(* IEC 61131-3 sources: mect_apps/TPAC1008_02_AB/RTU_test_PLC, 6 files *)

(* ---- Crosstable.gvl ---- *)
VAR_GLOBAL
errors_can AT %QD0.772:DINT;
errors_all AT %QD0.776:DINT;
min_latency_ms AT %QD0.780:DINT;
max_latency_ms AT %QD0.784:DINT;
Addr_node01 AT %IW0.800:UINT;
Life_node01 AT %IW0.804:UINT;
AnInCnf_1_node01 AT %QW0.808:UINT;
AnInCnf_2_node01 AT %QW0.812:UINT;
ValAi1_node01 AT %IW0.816:INT;
ValAi2_node01 AT %IW0.820:INT;
DigDir_1_node01 AT %QX0.824.0:BOOL;
DigDir_2_node01 AT %QX0.828.0:BOOL;
DigDir_3_node01 AT %QX0.832.0:BOOL;
DigDir_4_node01 AT %QX0.836.0:BOOL;
DigDir_5_node01 AT %QX0.840.0:BOOL;
DigDir_6_node01 AT %QX0.844.0:BOOL;
DigDir_7_node01 AT %QX0.848.0:BOOL;
DigDir_8_node01 AT %QX0.852.0:BOOL;
DigIn_2_node01 AT %IX0.856.0:BOOL;
DigIn_3_node01 AT %IX0.860.0:BOOL;
DigIn_6_node01 AT %IX0.864.0:BOOL;
DigIn_7_node01 AT %IX0.868.0:BOOL;
DigOut_1_node01 AT %QX0.872.0:BOOL;
DigOut_4_node01 AT %QX0.876.0:BOOL;
DigOut_5_node01 AT %QX0.880.0:BOOL;
DigOut_8_node01 AT %QX0.884.0:BOOL;
latency_01_ms AT %QD0.892:DINT;
min_latency_01_m AT %QD0.896:DINT;
max_latency_01_m AT %QD0.900:DINT;
errors_01 AT %QD0.908:DINT;
Addr_node02 AT %IW0.920:UINT;
Life_node02 AT %IW0.924:UINT;
AnInCnf_1_node02 AT %QW0.928:UINT;
AnInCnf_2_node02 AT %QW0.932:UINT;
ValAi1_node02 AT %IW0.936:INT;
ValAi2_node02 AT %IW0.940:INT;
DigDir_1_node02 AT %QX0.944.0:BOOL;
DigDir_2_node02 AT %QX0.948.0:BOOL;
DigDir_3_node02 AT %QX0.952.0:BOOL;
DigDir_4_node02 AT %QX0.956.0:BOOL;
DigDir_5_node02 AT %QX0.960.0:BOOL;
DigDir_6_node02 AT %QX0.964.0:BOOL;
DigDir_7_node02 AT %QX0.968.0:BOOL;
DigDir_8_node02 AT %QX0.972.0:BOOL;
DigIn_2_node02 AT %IX0.976.0:BOOL;
DigIn_3_node02 AT %IX0.980.0:BOOL;
DigIn_6_node02 AT %IX0.984.0:BOOL;
DigIn_7_node02 AT %IX0.988.0:BOOL;
DigOut_1_node02 AT %QX0.992.0:BOOL;
DigOut_4_node02 AT %QX0.996.0:BOOL;
DigOut_5_node02 AT %QX0.1000.0:BOOL;
DigOut_8_node02 AT %QX0.1004.0:BOOL;
latency_02_ms AT %QD0.1012:DINT;
min_latency_02_m AT %QD0.1016:DINT;
max_latency_02_m AT %QD0.1020:DINT;
errors_02 AT %QD0.1028:DINT;
Addr_node03 AT %IW0.1040:UINT;
Life_node03 AT %IW0.1044:UINT;
AnInCnf_1_node03 AT %QW0.1048:UINT;
AnInCnf_2_node03 AT %QW0.1052:UINT;
ValAi1_node03 AT %IW0.1056:INT;
ValAi2_node03 AT %IW0.1060:INT;
DigDir_1_node03 AT %QX0.1064.0:BOOL;
DigDir_2_node03 AT %QX0.1068.0:BOOL;
DigDir_3_node03 AT %QX0.1072.0:BOOL;
DigDir_4_node03 AT %QX0.1076.0:BOOL;
DigDir_5_node03 AT %QX0.1080.0:BOOL;
DigDir_6_node03 AT %QX0.1084.0:BOOL;
DigDir_7_node03 AT %QX0.1088.0:BOOL;
DigDir_8_node03 AT %QX0.1092.0:BOOL;
DigIn_2_node03 AT %IX0.1096.0:BOOL;
DigIn_3_node03 AT %IX0.1100.0:BOOL;
DigIn_6_node03 AT %IX0.1104.0:BOOL;
DigIn_7_node03 AT %IX0.1108.0:BOOL;
DigOut_1_node03 AT %QX0.1112.0:BOOL;
DigOut_4_node03 AT %QX0.1116.0:BOOL;
DigOut_5_node03 AT %QX0.1120.0:BOOL;
DigOut_8_node03 AT %QX0.1124.0:BOOL;
latency_03_ms AT %QD0.1132:DINT;
min_latency_03_m AT %QD0.1136:DINT;
max_latency_03_m AT %QD0.1140:DINT;
errors_03 AT %QD0.1148:DINT;
Addr_node04 AT %IW0.1160:UINT;
Life_node04 AT %IW0.1164:UINT;
AnInCnf_1_node04 AT %QW0.1168:UINT;
AnInCnf_2_node04 AT %QW0.1172:UINT;
ValAi1_node04 AT %IW0.1176:INT;
ValAi2_node04 AT %IW0.1180:INT;
DigDir_1_node04 AT %QX0.1184.0:BOOL;
DigDir_2_node04 AT %QX0.1188.0:BOOL;
DigDir_3_node04 AT %QX0.1192.0:BOOL;
DigDir_4_node04 AT %QX0.1196.0:BOOL;
DigDir_5_node04 AT %QX0.1200.0:BOOL;
DigDir_6_node04 AT %QX0.1204.0:BOOL;
DigDir_7_node04 AT %QX0.1208.0:BOOL;
DigDir_8_node04 AT %QX0.1212.0:BOOL;
DigIn_2_node04 AT %IX0.1216.0:BOOL;
DigIn_3_node04 AT %IX0.1220.0:BOOL;
DigIn_6_node04 AT %IX0.1224.0:BOOL;
DigIn_7_node04 AT %IX0.1228.0:BOOL;
DigOut_1_node04 AT %QX0.1232.0:BOOL;
DigOut_4_node04 AT %QX0.1236.0:BOOL;
DigOut_5_node04 AT %QX0.1240.0:BOOL;
DigOut_8_node04 AT %QX0.1244.0:BOOL;
latency_04_ms AT %QD0.1252:DINT;
min_latency_04_m AT %QD0.1256:DINT;
max_latency_04_m AT %QD0.1260:DINT;
errors_04 AT %QD0.1268:DINT;
Addr_node05 AT %IW0.1280:UINT;
Life_node05 AT %IW0.1284:UINT;
AnInCnf_1_node05 AT %QW0.1288:UINT;
AnInCnf_2_node05 AT %QW0.1292:UINT;
ValAi1_node05 AT %IW0.1296:INT;
ValAi2_node05 AT %IW0.1300:INT;
DigDir_1_node05 AT %QX0.1304.0:BOOL;
DigDir_2_node05 AT %QX0.1308.0:BOOL;
DigDir_3_node05 AT %QX0.1312.0:BOOL;
DigDir_4_node05 AT %QX0.1316.0:BOOL;
DigDir_5_node05 AT %QX0.1320.0:BOOL;
DigDir_6_node05 AT %QX0.1324.0:BOOL;
DigDir_7_node05 AT %QX0.1328.0:BOOL;
DigDir_8_node05 AT %QX0.1332.0:BOOL;
DigIn_2_node05 AT %IX0.1336.0:BOOL;
DigIn_3_node05 AT %IX0.1340.0:BOOL;
DigIn_6_node05 AT %IX0.1344.0:BOOL;
DigIn_7_node05 AT %IX0.1348.0:BOOL;
DigOut_1_node05 AT %QX0.1352.0:BOOL;
DigOut_4_node05 AT %QX0.1356.0:BOOL;
DigOut_5_node05 AT %QX0.1360.0:BOOL;
DigOut_8_node05 AT %QX0.1364.0:BOOL;
latency_05_ms AT %QD0.1372:DINT;
min_latency_05_m AT %QD0.1376:DINT;
max_latency_05_m AT %QD0.1380:DINT;
errors_05 AT %QD0.1388:DINT;
Addr_node06 AT %IW0.1400:UINT;
Life_node06 AT %IW0.1404:UINT;
AnInCnf_1_node06 AT %QW0.1408:UINT;
AnInCnf_2_node06 AT %QW0.1412:UINT;
ValAi1_node06 AT %IW0.1416:INT;
ValAi2_node06 AT %IW0.1420:INT;
DigDir_1_node06 AT %QX0.1424.0:BOOL;
DigDir_2_node06 AT %QX0.1428.0:BOOL;
DigDir_3_node06 AT %QX0.1432.0:BOOL;
DigDir_4_node06 AT %QX0.1436.0:BOOL;
DigDir_5_node06 AT %QX0.1440.0:BOOL;
DigDir_6_node06 AT %QX0.1444.0:BOOL;
DigDir_7_node06 AT %QX0.1448.0:BOOL;
DigDir_8_node06 AT %QX0.1452.0:BOOL;
DigIn_2_node06 AT %IX0.1456.0:BOOL;
DigIn_3_node06 AT %IX0.1460.0:BOOL;
DigIn_6_node06 AT %IX0.1464.0:BOOL;
DigIn_7_node06 AT %IX0.1468.0:BOOL;
DigOut_1_node06 AT %QX0.1472.0:BOOL;
DigOut_4_node06 AT %QX0.1476.0:BOOL;
DigOut_5_node06 AT %QX0.1480.0:BOOL;
DigOut_8_node06 AT %QX0.1484.0:BOOL;
latency_06_ms AT %QD0.1492:DINT;
min_latency_06_m AT %QD0.1496:DINT;
max_latency_06_m AT %QD0.1500:DINT;
errors_06 AT %QD0.1508:DINT;
Addr_node07 AT %IW0.1520:UINT;
Life_node07 AT %IW0.1524:UINT;
AnInCnf_1_node07 AT %QW0.1528:UINT;
AnInCnf_2_node07 AT %QW0.1532:UINT;
ValAi1_node07 AT %IW0.1536:INT;
ValAi2_node07 AT %IW0.1540:INT;
DigDir_1_node07 AT %QX0.1544.0:BOOL;
DigDir_2_node07 AT %QX0.1548.0:BOOL;
DigDir_3_node07 AT %QX0.1552.0:BOOL;
DigDir_4_node07 AT %QX0.1556.0:BOOL;
DigDir_5_node07 AT %QX0.1560.0:BOOL;
DigDir_6_node07 AT %QX0.1564.0:BOOL;
DigDir_7_node07 AT %QX0.1568.0:BOOL;
DigDir_8_node07 AT %QX0.1572.0:BOOL;
DigIn_2_node07 AT %IX0.1576.0:BOOL;
DigIn_3_node07 AT %IX0.1580.0:BOOL;
DigIn_6_node07 AT %IX0.1584.0:BOOL;
DigIn_7_node07 AT %IX0.1588.0:BOOL;
DigOut_1_node07 AT %QX0.1592.0:BOOL;
DigOut_4_node07 AT %QX0.1596.0:BOOL;
DigOut_5_node07 AT %QX0.1600.0:BOOL;
DigOut_8_node07 AT %QX0.1604.0:BOOL;
latency_07_ms AT %QD0.1612:DINT;
min_latency_07_m AT %QD0.1616:DINT;
max_latency_07_m AT %QD0.1620:DINT;
errors_07 AT %QD0.1628:DINT;
Addr_node08 AT %IW0.1640:UINT;
Life_node08 AT %IW0.1644:UINT;
AnInCnf_1_node08 AT %QW0.1648:UINT;
AnInCnf_2_node08 AT %QW0.1652:UINT;
ValAi1_node08 AT %IW0.1656:INT;
ValAi2_node08 AT %IW0.1660:INT;
DigDir_1_node08 AT %QX0.1664.0:BOOL;
DigDir_2_node08 AT %QX0.1668.0:BOOL;
DigDir_3_node08 AT %QX0.1672.0:BOOL;
DigDir_4_node08 AT %QX0.1676.0:BOOL;
DigDir_5_node08 AT %QX0.1680.0:BOOL;
DigDir_6_node08 AT %QX0.1684.0:BOOL;
DigDir_7_node08 AT %QX0.1688.0:BOOL;
DigDir_8_node08 AT %QX0.1692.0:BOOL;
DigIn_2_node08 AT %IX0.1696.0:BOOL;
DigIn_3_node08 AT %IX0.1700.0:BOOL;
DigIn_6_node08 AT %IX0.1704.0:BOOL;
DigIn_7_node08 AT %IX0.1708.0:BOOL;
DigOut_1_node08 AT %QX0.1712.0:BOOL;
DigOut_4_node08 AT %QX0.1716.0:BOOL;
DigOut_5_node08 AT %QX0.1720.0:BOOL;
DigOut_8_node08 AT %QX0.1724.0:BOOL;
latency_08_ms AT %QD0.1732:DINT;
min_latency_08_m AT %QD0.1736:DINT;
max_latency_08_m AT %QD0.1740:DINT;
errors_08 AT %QD0.1748:DINT;
Addr_node09 AT %IW0.1760:UINT;
Life_node09 AT %IW0.1764:UINT;
AnInCnf_1_node09 AT %QW0.1768:UINT;
AnInCnf_2_node09 AT %QW0.1772:UINT;
ValAi1_node09 AT %IW0.1776:INT;
ValAi2_node09 AT %IW0.1780:INT;
DigDir_1_node09 AT %QX0.1784.0:BOOL;
DigDir_2_node09 AT %QX0.1788.0:BOOL;
DigDir_3_node09 AT %QX0.1792.0:BOOL;
DigDir_4_node09 AT %QX0.1796.0:BOOL;
DigDir_5_node09 AT %QX0.1800.0:BOOL;
DigDir_6_node09 AT %QX0.1804.0:BOOL;
DigDir_7_node09 AT %QX0.1808.0:BOOL;
DigDir_8_node09 AT %QX0.1812.0:BOOL;
DigIn_2_node09 AT %IX0.1816.0:BOOL;
DigIn_3_node09 AT %IX0.1820.0:BOOL;
DigIn_6_node09 AT %IX0.1824.0:BOOL;
DigIn_7_node09 AT %IX0.1828.0:BOOL;
DigOut_1_node09 AT %QX0.1832.0:BOOL;
DigOut_4_node09 AT %QX0.1836.0:BOOL;
DigOut_5_node09 AT %QX0.1840.0:BOOL;
DigOut_8_node09 AT %QX0.1844.0:BOOL;
latency_09_ms AT %QD0.1852:DINT;
min_latency_09_m AT %QD0.1856:DINT;
max_latency_09_m AT %QD0.1860:DINT;
errors_09 AT %QD0.1868:DINT;
Addr_node10 AT %IW0.1880:UINT;
Life_node10 AT %IW0.1884:UINT;
AnInCnf_1_node10 AT %QW0.1888:UINT;
AnInCnf_2_node10 AT %QW0.1892:UINT;
ValAi1_node10 AT %IW0.1896:INT;
ValAi2_node10 AT %IW0.1900:INT;
DigDir_1_node10 AT %QX0.1904.0:BOOL;
DigDir_2_node10 AT %QX0.1908.0:BOOL;
DigDir_3_node10 AT %QX0.1912.0:BOOL;
DigDir_4_node10 AT %QX0.1916.0:BOOL;
DigDir_5_node10 AT %QX0.1920.0:BOOL;
DigDir_6_node10 AT %QX0.1924.0:BOOL;
DigDir_7_node10 AT %QX0.1928.0:BOOL;
DigDir_8_node10 AT %QX0.1932.0:BOOL;
DigIn_2_node10 AT %IX0.1936.0:BOOL;
DigIn_3_node10 AT %IX0.1940.0:BOOL;
DigIn_6_node10 AT %IX0.1944.0:BOOL;
DigIn_7_node10 AT %IX0.1948.0:BOOL;
DigOut_1_node10 AT %QX0.1952.0:BOOL;
DigOut_4_node10 AT %QX0.1956.0:BOOL;
DigOut_5_node10 AT %QX0.1960.0:BOOL;
DigOut_8_node10 AT %QX0.1964.0:BOOL;
latency_10_ms AT %QD0.1972:DINT;
min_latency_10_m AT %QD0.1976:DINT;
max_latency_10_m AT %QD0.1980:DINT;
errors_10 AT %QD0.1988:DINT;
Addr_node11 AT %IW0.2000:UINT;
Life_node11 AT %IW0.2004:UINT;
AnInCnf_1_node11 AT %QW0.2008:UINT;
AnInCnf_2_node11 AT %QW0.2012:UINT;
ValAi1_node11 AT %IW0.2016:INT;
ValAi2_node11 AT %IW0.2020:INT;
DigDir_1_node11 AT %QX0.2024.0:BOOL;
DigDir_2_node11 AT %QX0.2028.0:BOOL;
DigDir_3_node11 AT %QX0.2032.0:BOOL;
DigDir_4_node11 AT %QX0.2036.0:BOOL;
DigDir_5_node11 AT %QX0.2040.0:BOOL;
DigDir_6_node11 AT %QX0.2044.0:BOOL;
DigDir_7_node11 AT %QX0.2048.0:BOOL;
DigDir_8_node11 AT %QX0.2052.0:BOOL;
DigIn_2_node11 AT %IX0.2056.0:BOOL;
DigIn_3_node11 AT %IX0.2060.0:BOOL;
DigIn_6_node11 AT %IX0.2064.0:BOOL;
DigIn_7_node11 AT %IX0.2068.0:BOOL;
DigOut_1_node11 AT %QX0.2072.0:BOOL;
DigOut_4_node11 AT %QX0.2076.0:BOOL;
DigOut_5_node11 AT %QX0.2080.0:BOOL;
DigOut_8_node11 AT %QX0.2084.0:BOOL;
latency_11_ms AT %QD0.2092:DINT;
min_latency_11_m AT %QD0.2096:DINT;
max_latency_11_m AT %QD0.2100:DINT;
errors_11 AT %QD0.2108:DINT;
Addr_node12 AT %IW0.2120:UINT;
Life_node12 AT %IW0.2124:UINT;
AnInCnf_1_node12 AT %QW0.2128:UINT;
AnInCnf_2_node12 AT %QW0.2132:UINT;
ValAi1_node12 AT %IW0.2136:INT;
ValAi2_node12 AT %IW0.2140:INT;
DigDir_1_node12 AT %QX0.2144.0:BOOL;
DigDir_2_node12 AT %QX0.2148.0:BOOL;
DigDir_3_node12 AT %QX0.2152.0:BOOL;
DigDir_4_node12 AT %QX0.2156.0:BOOL;
DigDir_5_node12 AT %QX0.2160.0:BOOL;
DigDir_6_node12 AT %QX0.2164.0:BOOL;
DigDir_7_node12 AT %QX0.2168.0:BOOL;
DigDir_8_node12 AT %QX0.2172.0:BOOL;
DigIn_2_node12 AT %IX0.2176.0:BOOL;
DigIn_3_node12 AT %IX0.2180.0:BOOL;
DigIn_6_node12 AT %IX0.2184.0:BOOL;
DigIn_7_node12 AT %IX0.2188.0:BOOL;
DigOut_1_node12 AT %QX0.2192.0:BOOL;
DigOut_4_node12 AT %QX0.2196.0:BOOL;
DigOut_5_node12 AT %QX0.2200.0:BOOL;
DigOut_8_node12 AT %QX0.2204.0:BOOL;
latency_12_ms AT %QD0.2212:DINT;
min_latency_12_m AT %QD0.2216:DINT;
max_latency_12_m AT %QD0.2220:DINT;
errors_12 AT %QD0.2228:DINT;
Addr_node13 AT %IW0.2240:UINT;
Life_node13 AT %IW0.2244:UINT;
AnInCnf_1_node13 AT %QW0.2248:UINT;
AnInCnf_2_node13 AT %QW0.2252:UINT;
ValAi1_node13 AT %IW0.2256:INT;
ValAi2_node13 AT %IW0.2260:INT;
DigDir_1_node13 AT %QX0.2264.0:BOOL;
DigDir_2_node13 AT %QX0.2268.0:BOOL;
DigDir_3_node13 AT %QX0.2272.0:BOOL;
DigDir_4_node13 AT %QX0.2276.0:BOOL;
DigDir_5_node13 AT %QX0.2280.0:BOOL;
DigDir_6_node13 AT %QX0.2284.0:BOOL;
DigDir_7_node13 AT %QX0.2288.0:BOOL;
DigDir_8_node13 AT %QX0.2292.0:BOOL;
DigIn_2_node13 AT %IX0.2296.0:BOOL;
DigIn_3_node13 AT %IX0.2300.0:BOOL;
DigIn_6_node13 AT %IX0.2304.0:BOOL;
DigIn_7_node13 AT %IX0.2308.0:BOOL;
DigOut_1_node13 AT %QX0.2312.0:BOOL;
DigOut_4_node13 AT %QX0.2316.0:BOOL;
DigOut_5_node13 AT %QX0.2320.0:BOOL;
DigOut_8_node13 AT %QX0.2324.0:BOOL;
latency_13_ms AT %QD0.2332:DINT;
min_latency_13_m AT %QD0.2336:DINT;
max_latency_13_m AT %QD0.2340:DINT;
errors_13 AT %QD0.2348:DINT;
Addr_node14 AT %IW0.2360:UINT;
Life_node14 AT %IW0.2364:UINT;
AnInCnf_1_node14 AT %QW0.2368:UINT;
AnInCnf_2_node14 AT %QW0.2372:UINT;
ValAi1_node14 AT %IW0.2376:INT;
ValAi2_node14 AT %IW0.2380:INT;
DigDir_1_node14 AT %QX0.2384.0:BOOL;
DigDir_2_node14 AT %QX0.2388.0:BOOL;
DigDir_3_node14 AT %QX0.2392.0:BOOL;
DigDir_4_node14 AT %QX0.2396.0:BOOL;
DigDir_5_node14 AT %QX0.2400.0:BOOL;
DigDir_6_node14 AT %QX0.2404.0:BOOL;
DigDir_7_node14 AT %QX0.2408.0:BOOL;
DigDir_8_node14 AT %QX0.2412.0:BOOL;
DigIn_2_node14 AT %IX0.2416.0:BOOL;
DigIn_3_node14 AT %IX0.2420.0:BOOL;
DigIn_6_node14 AT %IX0.2424.0:BOOL;
DigIn_7_node14 AT %IX0.2428.0:BOOL;
DigOut_1_node14 AT %QX0.2432.0:BOOL;
DigOut_4_node14 AT %QX0.2436.0:BOOL;
DigOut_5_node14 AT %QX0.2440.0:BOOL;
DigOut_8_node14 AT %QX0.2444.0:BOOL;
latency_14_ms AT %QD0.2452:DINT;
min_latency_14_m AT %QD0.2456:DINT;
max_latency_14_m AT %QD0.2460:DINT;
errors_14 AT %QD0.2468:DINT;
Addr_node15 AT %IW0.2480:UINT;
Life_node15 AT %IW0.2484:UINT;
AnInCnf_1_node15 AT %QW0.2488:UINT;
AnInCnf_2_node15 AT %QW0.2492:UINT;
ValAi1_node15 AT %IW0.2496:INT;
ValAi2_node15 AT %IW0.2500:INT;
DigDir_1_node15 AT %QX0.2504.0:BOOL;
DigDir_2_node15 AT %QX0.2508.0:BOOL;
DigDir_3_node15 AT %QX0.2512.0:BOOL;
DigDir_4_node15 AT %QX0.2516.0:BOOL;
DigDir_5_node15 AT %QX0.2520.0:BOOL;
DigDir_6_node15 AT %QX0.2524.0:BOOL;
DigDir_7_node15 AT %QX0.2528.0:BOOL;
DigDir_8_node15 AT %QX0.2532.0:BOOL;
DigIn_2_node15 AT %IX0.2536.0:BOOL;
DigIn_3_node15 AT %IX0.2540.0:BOOL;
DigIn_6_node15 AT %IX0.2544.0:BOOL;
DigIn_7_node15 AT %IX0.2548.0:BOOL;
DigOut_1_node15 AT %QX0.2552.0:BOOL;
DigOut_4_node15 AT %QX0.2556.0:BOOL;
DigOut_5_node15 AT %QX0.2560.0:BOOL;
DigOut_8_node15 AT %QX0.2564.0:BOOL;
latency_15_ms AT %QD0.2572:DINT;
min_latency_15_m AT %QD0.2576:DINT;
max_latency_15_m AT %QD0.2580:DINT;
errors_15 AT %QD0.2588:DINT;
Addr_node16 AT %IW0.2600:UINT;
Life_node16 AT %IW0.2604:UINT;
AnInCnf_1_node16 AT %QW0.2608:UINT;
AnInCnf_2_node16 AT %QW0.2612:UINT;
ValAi1_node16 AT %IW0.2616:INT;
ValAi2_node16 AT %IW0.2620:INT;
DigDir_1_node16 AT %QX0.2624.0:BOOL;
DigDir_2_node16 AT %QX0.2628.0:BOOL;
DigDir_3_node16 AT %QX0.2632.0:BOOL;
DigDir_4_node16 AT %QX0.2636.0:BOOL;
DigDir_5_node16 AT %QX0.2640.0:BOOL;
DigDir_6_node16 AT %QX0.2644.0:BOOL;
DigDir_7_node16 AT %QX0.2648.0:BOOL;
DigDir_8_node16 AT %QX0.2652.0:BOOL;
DigIn_2_node16 AT %IX0.2656.0:BOOL;
DigIn_3_node16 AT %IX0.2660.0:BOOL;
DigIn_6_node16 AT %IX0.2664.0:BOOL;
DigIn_7_node16 AT %IX0.2668.0:BOOL;
DigOut_1_node16 AT %QX0.2672.0:BOOL;
DigOut_4_node16 AT %QX0.2676.0:BOOL;
DigOut_5_node16 AT %QX0.2680.0:BOOL;
DigOut_8_node16 AT %QX0.2684.0:BOOL;
latency_16_ms AT %QD0.2692:DINT;
min_latency_16_m AT %QD0.2696:DINT;
max_latency_16_m AT %QD0.2700:DINT;
errors_16 AT %QD0.2708:DINT;
Addr_node17 AT %IW0.2720:UINT;
Life_node17 AT %IW0.2724:UINT;
AnInCnf_1_node17 AT %QW0.2728:UINT;
AnInCnf_2_node17 AT %QW0.2732:UINT;
ValAi1_node17 AT %IW0.2736:INT;
ValAi2_node17 AT %IW0.2740:INT;
DigDir_1_node17 AT %QX0.2744.0:BOOL;
DigDir_2_node17 AT %QX0.2748.0:BOOL;
DigDir_3_node17 AT %QX0.2752.0:BOOL;
DigDir_4_node17 AT %QX0.2756.0:BOOL;
DigDir_5_node17 AT %QX0.2760.0:BOOL;
DigDir_6_node17 AT %QX0.2764.0:BOOL;
DigDir_7_node17 AT %QX0.2768.0:BOOL;
DigDir_8_node17 AT %QX0.2772.0:BOOL;
DigIn_2_node17 AT %IX0.2776.0:BOOL;
DigIn_3_node17 AT %IX0.2780.0:BOOL;
DigIn_6_node17 AT %IX0.2784.0:BOOL;
DigIn_7_node17 AT %IX0.2788.0:BOOL;
DigOut_1_node17 AT %QX0.2792.0:BOOL;
DigOut_4_node17 AT %QX0.2796.0:BOOL;
DigOut_5_node17 AT %QX0.2800.0:BOOL;
DigOut_8_node17 AT %QX0.2804.0:BOOL;
latency_17_ms AT %QD0.2812:DINT;
min_latency_17_m AT %QD0.2816:DINT;
max_latency_17_m AT %QD0.2820:DINT;
errors_17 AT %QD0.2828:DINT;
Addr_node18 AT %IW0.2840:UINT;
Life_node18 AT %IW0.2844:UINT;
AnInCnf_1_node18 AT %QW0.2848:UINT;
AnInCnf_2_node18 AT %QW0.2852:UINT;
ValAi1_node18 AT %IW0.2856:INT;
ValAi2_node18 AT %IW0.2860:INT;
DigDir_1_node18 AT %QX0.2864.0:BOOL;
DigDir_2_node18 AT %QX0.2868.0:BOOL;
DigDir_3_node18 AT %QX0.2872.0:BOOL;
DigDir_4_node18 AT %QX0.2876.0:BOOL;
DigDir_5_node18 AT %QX0.2880.0:BOOL;
DigDir_6_node18 AT %QX0.2884.0:BOOL;
DigDir_7_node18 AT %QX0.2888.0:BOOL;
DigDir_8_node18 AT %QX0.2892.0:BOOL;
DigIn_2_node18 AT %IX0.2896.0:BOOL;
DigIn_3_node18 AT %IX0.2900.0:BOOL;
DigIn_6_node18 AT %IX0.2904.0:BOOL;
DigIn_7_node18 AT %IX0.2908.0:BOOL;
DigOut_1_node18 AT %QX0.2912.0:BOOL;
DigOut_4_node18 AT %QX0.2916.0:BOOL;
DigOut_5_node18 AT %QX0.2920.0:BOOL;
DigOut_8_node18 AT %QX0.2924.0:BOOL;
latency_18_ms AT %QD0.2932:DINT;
min_latency_18_m AT %QD0.2936:DINT;
max_latency_18_m AT %QD0.2940:DINT;
errors_18 AT %QD0.2948:DINT;
Addr_node19 AT %IW0.2960:UINT;
Life_node19 AT %IW0.2964:UINT;
AnInCnf_1_node19 AT %QW0.2968:UINT;
AnInCnf_2_node19 AT %QW0.2972:UINT;
ValAi1_node19 AT %IW0.2976:INT;
ValAi2_node19 AT %IW0.2980:INT;
DigDir_1_node19 AT %QX0.2984.0:BOOL;
DigDir_2_node19 AT %QX0.2988.0:BOOL;
DigDir_3_node19 AT %QX0.2992.0:BOOL;
DigDir_4_node19 AT %QX0.2996.0:BOOL;
DigDir_5_node19 AT %QX0.3000.0:BOOL;
DigDir_6_node19 AT %QX0.3004.0:BOOL;
DigDir_7_node19 AT %QX0.3008.0:BOOL;
DigDir_8_node19 AT %QX0.3012.0:BOOL;
DigIn_2_node19 AT %IX0.3016.0:BOOL;
DigIn_3_node19 AT %IX0.3020.0:BOOL;
DigIn_6_node19 AT %IX0.3024.0:BOOL;
DigIn_7_node19 AT %IX0.3028.0:BOOL;
DigOut_1_node19 AT %QX0.3032.0:BOOL;
DigOut_4_node19 AT %QX0.3036.0:BOOL;
DigOut_5_node19 AT %QX0.3040.0:BOOL;
DigOut_8_node19 AT %QX0.3044.0:BOOL;
latency_19_ms AT %QD0.3052:DINT;
min_latency_19_m AT %QD0.3056:DINT;
max_latency_19_m AT %QD0.3060:DINT;
errors_19 AT %QD0.3068:DINT;
Addr_node20 AT %IW0.3080:UINT;
Life_node20 AT %IW0.3084:UINT;
AnInCnf_1_node20 AT %QW0.3088:UINT;
AnInCnf_2_node20 AT %QW0.3092:UINT;
ValAi1_node20 AT %IW0.3096:INT;
ValAi2_node20 AT %IW0.3100:INT;
DigDir_1_node20 AT %QX0.3104.0:BOOL;
DigDir_2_node20 AT %QX0.3108.0:BOOL;
DigDir_3_node20 AT %QX0.3112.0:BOOL;
DigDir_4_node20 AT %QX0.3116.0:BOOL;
DigDir_5_node20 AT %QX0.3120.0:BOOL;
DigDir_6_node20 AT %QX0.3124.0:BOOL;
DigDir_7_node20 AT %QX0.3128.0:BOOL;
DigDir_8_node20 AT %QX0.3132.0:BOOL;
DigIn_2_node20 AT %IX0.3136.0:BOOL;
DigIn_3_node20 AT %IX0.3140.0:BOOL;
DigIn_6_node20 AT %IX0.3144.0:BOOL;
DigIn_7_node20 AT %IX0.3148.0:BOOL;
DigOut_1_node20 AT %QX0.3152.0:BOOL;
DigOut_4_node20 AT %QX0.3156.0:BOOL;
DigOut_5_node20 AT %QX0.3160.0:BOOL;
DigOut_8_node20 AT %QX0.3164.0:BOOL;
latency_20_ms AT %QD0.3172:DINT;
min_latency_20_m AT %QD0.3176:DINT;
max_latency_20_m AT %QD0.3180:DINT;
errors_20 AT %QD0.3188:DINT;
Addr_node21 AT %IW0.3200:UINT;
Life_node21 AT %IW0.3204:UINT;
AnInCnf_1_node21 AT %QW0.3208:UINT;
AnInCnf_2_node21 AT %QW0.3212:UINT;
ValAi1_node21 AT %IW0.3216:INT;
ValAi2_node21 AT %IW0.3220:INT;
DigDir_1_node21 AT %QX0.3224.0:BOOL;
DigDir_2_node21 AT %QX0.3228.0:BOOL;
DigDir_3_node21 AT %QX0.3232.0:BOOL;
DigDir_4_node21 AT %QX0.3236.0:BOOL;
DigDir_5_node21 AT %QX0.3240.0:BOOL;
DigDir_6_node21 AT %QX0.3244.0:BOOL;
DigDir_7_node21 AT %QX0.3248.0:BOOL;
DigDir_8_node21 AT %QX0.3252.0:BOOL;
DigIn_2_node21 AT %IX0.3256.0:BOOL;
DigIn_3_node21 AT %IX0.3260.0:BOOL;
DigIn_6_node21 AT %IX0.3264.0:BOOL;
DigIn_7_node21 AT %IX0.3268.0:BOOL;
DigOut_1_node21 AT %QX0.3272.0:BOOL;
DigOut_4_node21 AT %QX0.3276.0:BOOL;
DigOut_5_node21 AT %QX0.3280.0:BOOL;
DigOut_8_node21 AT %QX0.3284.0:BOOL;
latency_21_ms AT %QD0.3292:DINT;
min_latency_21_m AT %QD0.3296:DINT;
max_latency_21_m AT %QD0.3300:DINT;
errors_21 AT %QD0.3308:DINT;
Addr_node22 AT %IW0.3320:UINT;
Life_node22 AT %IW0.3324:UINT;
AnInCnf_1_node22 AT %QW0.3328:UINT;
AnInCnf_2_node22 AT %QW0.3332:UINT;
ValAi1_node22 AT %IW0.3336:INT;
ValAi2_node22 AT %IW0.3340:INT;
DigDir_1_node22 AT %QX0.3344.0:BOOL;
DigDir_2_node22 AT %QX0.3348.0:BOOL;
DigDir_3_node22 AT %QX0.3352.0:BOOL;
DigDir_4_node22 AT %QX0.3356.0:BOOL;
DigDir_5_node22 AT %QX0.3360.0:BOOL;
DigDir_6_node22 AT %QX0.3364.0:BOOL;
DigDir_7_node22 AT %QX0.3368.0:BOOL;
DigDir_8_node22 AT %QX0.3372.0:BOOL;
DigIn_2_node22 AT %IX0.3376.0:BOOL;
DigIn_3_node22 AT %IX0.3380.0:BOOL;
DigIn_6_node22 AT %IX0.3384.0:BOOL;
DigIn_7_node22 AT %IX0.3388.0:BOOL;
DigOut_1_node22 AT %QX0.3392.0:BOOL;
DigOut_4_node22 AT %QX0.3396.0:BOOL;
DigOut_5_node22 AT %QX0.3400.0:BOOL;
DigOut_8_node22 AT %QX0.3404.0:BOOL;
latency_22_ms AT %QD0.3412:DINT;
min_latency_22_m AT %QD0.3416:DINT;
max_latency_22_m AT %QD0.3420:DINT;
errors_22 AT %QD0.3428:DINT;
Addr_node23 AT %IW0.3440:UINT;
Life_node23 AT %IW0.3444:UINT;
AnInCnf_1_node23 AT %QW0.3448:UINT;
AnInCnf_2_node23 AT %QW0.3452:UINT;
ValAi1_node23 AT %IW0.3456:INT;
ValAi2_node23 AT %IW0.3460:INT;
DigDir_1_node23 AT %QX0.3464.0:BOOL;
DigDir_2_node23 AT %QX0.3468.0:BOOL;
DigDir_3_node23 AT %QX0.3472.0:BOOL;
DigDir_4_node23 AT %QX0.3476.0:BOOL;
DigDir_5_node23 AT %QX0.3480.0:BOOL;
DigDir_6_node23 AT %QX0.3484.0:BOOL;
DigDir_7_node23 AT %QX0.3488.0:BOOL;
DigDir_8_node23 AT %QX0.3492.0:BOOL;
DigIn_2_node23 AT %IX0.3496.0:BOOL;
DigIn_3_node23 AT %IX0.3500.0:BOOL;
DigIn_6_node23 AT %IX0.3504.0:BOOL;
DigIn_7_node23 AT %IX0.3508.0:BOOL;
DigOut_1_node23 AT %QX0.3512.0:BOOL;
DigOut_4_node23 AT %QX0.3516.0:BOOL;
DigOut_5_node23 AT %QX0.3520.0:BOOL;
DigOut_8_node23 AT %QX0.3524.0:BOOL;
latency_23_ms AT %QD0.3532:DINT;
min_latency_23_m AT %QD0.3536:DINT;
max_latency_23_m AT %QD0.3540:DINT;
errors_23 AT %QD0.3548:DINT;
Addr_node24 AT %IW0.3560:UINT;
Life_node24 AT %IW0.3564:UINT;
AnInCnf_1_node24 AT %QW0.3568:UINT;
AnInCnf_2_node24 AT %QW0.3572:UINT;
ValAi1_node24 AT %IW0.3576:INT;
ValAi2_node24 AT %IW0.3580:INT;
DigDir_1_node24 AT %QX0.3584.0:BOOL;
DigDir_2_node24 AT %QX0.3588.0:BOOL;
DigDir_3_node24 AT %QX0.3592.0:BOOL;
DigDir_4_node24 AT %QX0.3596.0:BOOL;
DigDir_5_node24 AT %QX0.3600.0:BOOL;
DigDir_6_node24 AT %QX0.3604.0:BOOL;
DigDir_7_node24 AT %QX0.3608.0:BOOL;
DigDir_8_node24 AT %QX0.3612.0:BOOL;
DigIn_2_node24 AT %IX0.3616.0:BOOL;
DigIn_3_node24 AT %IX0.3620.0:BOOL;
DigIn_6_node24 AT %IX0.3624.0:BOOL;
DigIn_7_node24 AT %IX0.3628.0:BOOL;
DigOut_1_node24 AT %QX0.3632.0:BOOL;
DigOut_4_node24 AT %QX0.3636.0:BOOL;
DigOut_5_node24 AT %QX0.3640.0:BOOL;
DigOut_8_node24 AT %QX0.3644.0:BOOL;
latency_24_ms AT %QD0.3652:DINT;
min_latency_24_m AT %QD0.3656:DINT;
max_latency_24_m AT %QD0.3660:DINT;
errors_24 AT %QD0.3668:DINT;
RTU0_TYPE_PORT AT %ID0.20000:UDINT;
RTU0_BAUDRATE AT %ID0.20004:UDINT;
RTU0_STATUS AT %ID0.20008:UDINT;
RTU0_READS AT %ID0.20012:UDINT;
RTU0_WRITES AT %ID0.20016:UDINT;
RTU0_TIMEOUTS AT %ID0.20020:UDINT;
RTU0_COMM_ERRORS AT %ID0.20024:UDINT;
RTU0_LAST_ERROR AT %ID0.20028:UDINT;
RTU0_WRITE_QUEUE AT %ID0.20032:UDINT;
RTU0_READ_QUEUE AT %ID0.20036:UDINT;
RTU1_TYPE_PORT AT %ID0.20040:UDINT;
RTU1_BAUDRATE AT %ID0.20044:UDINT;
RTU1_STATUS AT %ID0.20048:UDINT;
RTU1_READS AT %ID0.20052:UDINT;
RTU1_WRITES AT %ID0.20056:UDINT;
RTU1_TIMEOUTS AT %ID0.20060:UDINT;
RTU1_COMM_ERRORS AT %ID0.20064:UDINT;
RTU1_LAST_ERROR AT %ID0.20068:UDINT;
RTU1_WRITE_QUEUE AT %ID0.20072:UDINT;
RTU1_READ_QUEUE AT %ID0.20076:UDINT;
RTU3_TYPE_PORT AT %ID0.20080:UDINT;
RTU3_BAUDRATE AT %ID0.20084:UDINT;
RTU3_STATUS AT %ID0.20088:UDINT;
RTU3_READS AT %ID0.20092:UDINT;
RTU3_WRITES AT %ID0.20096:UDINT;
RTU3_TIMEOUTS AT %ID0.20100:UDINT;
RTU3_COMM_ERRORS AT %ID0.20104:UDINT;
RTU3_LAST_ERROR AT %ID0.20108:UDINT;
RTU3_WRITE_QUEUE AT %ID0.20112:UDINT;
RTU3_READ_QUEUE AT %ID0.20116:UDINT;
CAN0_TYPE_PORT AT %ID0.20120:UDINT;
CAN0_BAUDRATE AT %ID0.20124:UDINT;
CAN0_STATUS AT %ID0.20128:UDINT;
CAN0_READS AT %ID0.20132:UDINT;
CAN0_WRITES AT %ID0.20136:UDINT;
CAN0_TIMEOUTS AT %ID0.20140:UDINT;
CAN0_COMM_ERRORS AT %ID0.20144:UDINT;
CAN0_LAST_ERROR AT %ID0.20148:UDINT;
CAN0_WRITE_QUEUE AT %ID0.20152:UDINT;
CAN0_READ_QUEUE AT %ID0.20156:UDINT;
CAN1_TYPE_PORT AT %ID0.20160:UDINT;
CAN1_BAUDRATE AT %ID0.20164:UDINT;
CAN1_STATUS AT %ID0.20168:UDINT;
CAN1_READS AT %ID0.20172:UDINT;
CAN1_WRITES AT %ID0.20176:UDINT;
CAN1_TIMEOUTS AT %ID0.20180:UDINT;
CAN1_COMM_ERRORS AT %ID0.20184:UDINT;
CAN1_LAST_ERROR AT %ID0.20188:UDINT;
CAN1_WRITE_QUEUE AT %ID0.20192:UDINT;
CAN1_READ_QUEUE AT %ID0.20196:UDINT;
TCPS_TYPE_PORT AT %ID0.20200:UDINT;
TCPS_IP_ADDRESS AT %ID0.20204:UDINT;
TCPS_STATUS AT %ID0.20208:UDINT;
TCPS_READS AT %ID0.20212:UDINT;
TCPS_WRITES AT %ID0.20216:UDINT;
TCPS_TIMEOUTS AT %ID0.20220:UDINT;
TCPS_COMM_ERRORS AT %ID0.20224:UDINT;
TCPS_LAST_ERROR AT %ID0.20228:UDINT;
TCPS_WRITE_QUEUE AT %ID0.20232:UDINT;
TCPS_READ_QUEUE AT %ID0.20236:UDINT;
TCP0_TYPE_PORT AT %ID0.20240:UDINT;
TCP0_IP_ADDRESS AT %ID0.20244:UDINT;
TCP0_STATUS AT %ID0.20248:UDINT;
TCP0_READS AT %ID0.20252:UDINT;
TCP0_WRITES AT %ID0.20256:UDINT;
TCP0_TIMEOUTS AT %ID0.20260:UDINT;
TCP0_COMM_ERRORS AT %ID0.20264:UDINT;
TCP0_LAST_ERROR AT %ID0.20268:UDINT;
TCP0_WRITE_QUEUE AT %ID0.20272:UDINT;
TCP0_READ_QUEUE AT %ID0.20276:UDINT;
TCP1_TYPE_PORT AT %ID0.20280:UDINT;
TCP1_IP_ADDRESS AT %ID0.20284:UDINT;
TCP1_STATUS AT %ID0.20288:UDINT;
TCP1_READS AT %ID0.20292:UDINT;
TCP1_WRITES AT %ID0.20296:UDINT;
TCP1_TIMEOUTS AT %ID0.20300:UDINT;
TCP1_COMM_ERRORS AT %ID0.20304:UDINT;
TCP1_LAST_ERROR AT %ID0.20308:UDINT;
TCP1_WRITE_QUEUE AT %ID0.20312:UDINT;
TCP1_READ_QUEUE AT %ID0.20316:UDINT;
TCP2_TYPE_PORT AT %ID0.20320:UDINT;
TCP2_IP_ADDRESS AT %ID0.20324:UDINT;
TCP2_STATUS AT %ID0.20328:UDINT;
TCP2_READS AT %ID0.20332:UDINT;
TCP2_WRITES AT %ID0.20336:UDINT;
TCP2_TIMEOUTS AT %ID0.20340:UDINT;
TCP2_COMM_ERRORS AT %ID0.20344:UDINT;
TCP2_LAST_ERROR AT %ID0.20348:UDINT;
TCP2_WRITE_QUEUE AT %ID0.20352:UDINT;
TCP2_READ_QUEUE AT %ID0.20356:UDINT;
TCP3_TYPE_PORT AT %ID0.20360:UDINT;
TCP3_IP_ADDRESS AT %ID0.20364:UDINT;
TCP3_STATUS AT %ID0.20368:UDINT;
TCP3_READS AT %ID0.20372:UDINT;
TCP3_WRITES AT %ID0.20376:UDINT;
TCP3_TIMEOUTS AT %ID0.20380:UDINT;
TCP3_COMM_ERRORS AT %ID0.20384:UDINT;
TCP3_LAST_ERROR AT %ID0.20388:UDINT;
TCP3_WRITE_QUEUE AT %ID0.20392:UDINT;
TCP3_READ_QUEUE AT %ID0.20396:UDINT;
TCP4_TYPE_PORT AT %ID0.20400:UDINT;
TCP4_IP_ADDRESS AT %ID0.20404:UDINT;
TCP4_STATUS AT %ID0.20408:UDINT;
TCP4_READS AT %ID0.20412:UDINT;
TCP4_WRITES AT %ID0.20416:UDINT;
TCP4_TIMEOUTS AT %ID0.20420:UDINT;
TCP4_COMM_ERRORS AT %ID0.20424:UDINT;
TCP4_LAST_ERROR AT %ID0.20428:UDINT;
TCP4_WRITE_QUEUE AT %ID0.20432:UDINT;
TCP4_READ_QUEUE AT %ID0.20436:UDINT;
TCP5_TYPE_PORT AT %ID0.20440:UDINT;
TCP5_IP_ADDRESS AT %ID0.20444:UDINT;
TCP5_STATUS AT %ID0.20448:UDINT;
TCP5_READS AT %ID0.20452:UDINT;
TCP5_WRITES AT %ID0.20456:UDINT;
TCP5_TIMEOUTS AT %ID0.20460:UDINT;
TCP5_COMM_ERRORS AT %ID0.20464:UDINT;
TCP5_LAST_ERROR AT %ID0.20468:UDINT;
TCP5_WRITE_QUEUE AT %ID0.20472:UDINT;
TCP5_READ_QUEUE AT %ID0.20476:UDINT;
TCP6_TYPE_PORT AT %ID0.20480:UDINT;
TCP6_IP_ADDRESS AT %ID0.20484:UDINT;
TCP6_STATUS AT %ID0.20488:UDINT;
TCP6_READS AT %ID0.20492:UDINT;
TCP6_WRITES AT %ID0.20496:UDINT;
TCP6_TIMEOUTS AT %ID0.20500:UDINT;
TCP6_COMM_ERRORS AT %ID0.20504:UDINT;
TCP6_LAST_ERROR AT %ID0.20508:UDINT;
TCP6_WRITE_QUEUE AT %ID0.20512:UDINT;
TCP6_READ_QUEUE AT %ID0.20516:UDINT;
TCP7_TYPE_PORT AT %ID0.20520:UDINT;
TCP7_IP_ADDRESS AT %ID0.20524:UDINT;
TCP7_STATUS AT %ID0.20528:UDINT;
TCP7_READS AT %ID0.20532:UDINT;
TCP7_WRITES AT %ID0.20536:UDINT;
TCP7_TIMEOUTS AT %ID0.20540:UDINT;
TCP7_COMM_ERRORS AT %ID0.20544:UDINT;
TCP7_LAST_ERROR AT %ID0.20548:UDINT;
TCP7_WRITE_QUEUE AT %ID0.20552:UDINT;
TCP7_READ_QUEUE AT %ID0.20556:UDINT;
TCP8_TYPE_PORT AT %ID0.20560:UDINT;
TCP8_IP_ADDRESS AT %ID0.20564:UDINT;
TCP8_STATUS AT %ID0.20568:UDINT;
TCP8_READS AT %ID0.20572:UDINT;
TCP8_WRITES AT %ID0.20576:UDINT;
TCP8_TIMEOUTS AT %ID0.20580:UDINT;
TCP8_COMM_ERRORS AT %ID0.20584:UDINT;
TCP8_LAST_ERROR AT %ID0.20588:UDINT;
TCP8_WRITE_QUEUE AT %ID0.20592:UDINT;
TCP8_READ_QUEUE AT %ID0.20596:UDINT;
TCP9_TYPE_PORT AT %ID0.20600:UDINT;
TCP9_IP_ADDRESS AT %ID0.20604:UDINT;
TCP9_STATUS AT %ID0.20608:UDINT;
TCP9_READS AT %ID0.20612:UDINT;
TCP9_WRITES AT %ID0.20616:UDINT;
TCP9_TIMEOUTS AT %ID0.20620:UDINT;
TCP9_COMM_ERRORS AT %ID0.20624:UDINT;
TCP9_LAST_ERROR AT %ID0.20628:UDINT;
TCP9_WRITE_QUEUE AT %ID0.20632:UDINT;
TCP9_READ_QUEUE AT %ID0.20636:UDINT;
NODE_01_DEV_NODE AT %ID0.20688:UDINT;
NODE_01_STATUS AT %ID0.20692:UDINT;
NODE_02_DEV_NODE AT %ID0.20696:UDINT;
NODE_02_STATUS AT %ID0.20700:UDINT;
NODE_03_DEV_NODE AT %ID0.20704:UDINT;
NODE_03_STATUS AT %ID0.20708:UDINT;
NODE_04_DEV_NODE AT %ID0.20712:UDINT;
NODE_04_STATUS AT %ID0.20716:UDINT;
NODE_05_DEV_NODE AT %ID0.20720:UDINT;
NODE_05_STATUS AT %ID0.20724:UDINT;
NODE_06_DEV_NODE AT %ID0.20728:UDINT;
NODE_06_STATUS AT %ID0.20732:UDINT;
NODE_07_DEV_NODE AT %ID0.20736:UDINT;
NODE_07_STATUS AT %ID0.20740:UDINT;
NODE_08_DEV_NODE AT %ID0.20744:UDINT;
NODE_08_STATUS AT %ID0.20748:UDINT;
NODE_09_DEV_NODE AT %ID0.20752:UDINT;
NODE_09_STATUS AT %ID0.20756:UDINT;
NODE_10_DEV_NODE AT %ID0.20760:UDINT;
NODE_10_STATUS AT %ID0.20764:UDINT;
NODE_11_DEV_NODE AT %ID0.20768:UDINT;
NODE_11_STATUS AT %ID0.20772:UDINT;
NODE_12_DEV_NODE AT %ID0.20776:UDINT;
NODE_12_STATUS AT %ID0.20780:UDINT;
NODE_13_DEV_NODE AT %ID0.20784:UDINT;
NODE_13_STATUS AT %ID0.20788:UDINT;
NODE_14_DEV_NODE AT %ID0.20792:UDINT;
NODE_14_STATUS AT %ID0.20796:UDINT;
NODE_15_DEV_NODE AT %ID0.20800:UDINT;
NODE_15_STATUS AT %ID0.20804:UDINT;
NODE_16_DEV_NODE AT %ID0.20808:UDINT;
NODE_16_STATUS AT %ID0.20812:UDINT;
NODE_17_DEV_NODE AT %ID0.20816:UDINT;
NODE_17_STATUS AT %ID0.20820:UDINT;
NODE_18_DEV_NODE AT %ID0.20824:UDINT;
NODE_18_STATUS AT %ID0.20828:UDINT;
NODE_19_DEV_NODE AT %ID0.20832:UDINT;
NODE_19_STATUS AT %ID0.20836:UDINT;
NODE_20_DEV_NODE AT %ID0.20840:UDINT;
NODE_20_STATUS AT %ID0.20844:UDINT;
NODE_21_DEV_NODE AT %ID0.20848:UDINT;
NODE_21_STATUS AT %ID0.20852:UDINT;
NODE_22_DEV_NODE AT %ID0.20856:UDINT;
NODE_22_STATUS AT %ID0.20860:UDINT;
NODE_23_DEV_NODE AT %ID0.20864:UDINT;
NODE_23_STATUS AT %ID0.20868:UDINT;
NODE_24_DEV_NODE AT %ID0.20872:UDINT;
NODE_24_STATUS AT %ID0.20876:UDINT;
PLC_DigIn_1 AT %IX0.21200.0:BOOL;
PLC_DigIn_2 AT %IX0.21204.0:BOOL;
PLC_DigIn_3 AT %IX0.21208.0:BOOL;
PLC_DigIn_4 AT %IX0.21212.0:BOOL;
PLC_DigIn_5 AT %IX0.21216.0:BOOL;
PLC_DigIn_6 AT %IX0.21220.0:BOOL;
PLC_DigIn_7 AT %IX0.21224.0:BOOL;
PLC_DigIn_8 AT %IX0.21228.0:BOOL;
PLC_Reserved_1 AT %IX0.21232.0:BOOL;
PLC_DigOut_1 AT %QX0.21236.0:BOOL;
PLC_DigOut_2 AT %QX0.21240.0:BOOL;
PLC_DigOut_3 AT %QX0.21244.0:BOOL;
PLC_DigOut_4 AT %QX0.21248.0:BOOL;
PLC_DigOut_5 AT %QX0.21252.0:BOOL;
PLC_DigOut_6 AT %QX0.21256.0:BOOL;
PLC_DigOut_7 AT %QX0.21260.0:BOOL;
PLC_DigOut_8 AT %QX0.21264.0:BOOL;
PLC_DigOut_9 AT %QX0.21268.0:BOOL;
PLC_DigOut_10 AT %QX0.21272.0:BOOL;
PLC_DigOut_11 AT %QX0.21276.0:BOOL;
PLC_DigOut_12 AT %QX0.21280.0:BOOL;
PLC_Hwconf AT %IW0.21284:UINT;
PLC_Revisione AT %IW0.21288:UINT;
PLC_StatusReg AT %IW0.21292:UINT;
PLC_Heartbeat AT %IW0.21296:UINT;
PLC_AnIn_1 AT %IW0.21300:INT;
PLC_AnIn_2 AT %IW0.21304:INT;
PLC_AnIn_3 AT %IW0.21308:INT;
PLC_AnIn_4 AT %IW0.21312:INT;
PLC_EncoderCo_Lo AT %IW0.21316:UINT;
PLC_EncoderCo_Hi AT %IW0.21320:UINT;
PLC_CaptureT1_Lo AT %IW0.21324:UINT;
PLC_CaptureT1_Hi AT %IW0.21328:UINT;
PLC_CaptureT2_Lo AT %IW0.21332:UINT;
PLC_CaptureT2_Hi AT %IW0.21336:UINT;
PLC_RPM AT %IW0.21340:UINT;
PLC_Tamb AT %IW0.21344:INT;
PLC_EnableEnc AT %QW0.21348:UINT;
PLC_ResetCount AT %QW0.21352:UINT;
PLC_AnInConf_1 AT %QW0.21356:UINT;
PLC_AnInConf_2 AT %QW0.21360:UINT;
PLC_AnInConf_3 AT %QW0.21364:UINT;
PLC_AnInConf_4 AT %QW0.21368:UINT;
PLC_AnOutConf_1 AT %QW0.21372:UINT;
PLC_AnOutConf_2 AT %QW0.21376:UINT;
PLC_Reserved_2 AT %QW0.21380:UINT;
PLC_Reserved_3 AT %QW0.21384:UINT;
PLC_AnOut_1 AT %QW0.21388:INT;
PLC_AnOut_2 AT %QW0.21392:INT;
PLC_Reserved_4 AT %QW0.21396:INT;
PLC_Reserved_5 AT %QW0.21400:INT;
PLC_FiltAnIn_1 AT %QW0.21404:UINT;
PLC_FiltAnIn_2 AT %QW0.21408:UINT;
PLC_FiltAnIn_3 AT %QW0.21412:UINT;
PLC_FiltAnIn_4 AT %QW0.21416:UINT;
CH0_NETRUN AT %IX0.21428.0:BOOL;
CH0_NETGOOD AT %IX0.21432.0:BOOL;
CH0_NETERR AT %ID0.21436:UDINT;
CH0_NETRST AT %QX0.21440.0:BOOL;
CH0_NETDIS AT %QX0.21444.0:BOOL;
CH0_01_NODERUN AT %IX0.21448.0:BOOL;
CH0_01_NODEGOOD AT %IX0.21452.0:BOOL;
CH0_01_NODEERR AT %ID0.21456:UDINT;
CH0_01_NODERST AT %QX0.21460.0:BOOL;
CH0_01_NODEDIS AT %QX0.21464.0:BOOL;
PLC_time AT %ID0.21560:REAL;
PLC_timeMin AT %ID0.21564:REAL;
PLC_timeMax AT %ID0.21568:REAL;
PLC_timeWin AT %QD0.21572:REAL;
PLC_Version AT %IW0.21576:UINT;
PLC_EngineStatus AT %IW0.21580:UINT;
PLC_ResetValues AT %QX0.21584.0:BOOL;
PLC_buzzerOn AT %QX0.21588.0:BOOL;
END_VAR

(* ---- set_min_dint.st ---- *)
(*[[
]]*)
FUNCTION set_min_dint
VAR_IN_OUT
    A : DINT;
END_VAR
VAR_INPUT
    B : DINT;
END_VAR

	if A < 0 or B < A then
		A := B;
	end_if;

END_FUNCTION

(* ---- Fast.st ---- *)
(*[[
]]*)
PROGRAM Fast
#import "Crosstable.gvl"
#import "Resource1.gvl"
VAR

END_VAR

;

END_PROGRAM

(* ---- Init.st ---- *)
(*[[
]]*)
PROGRAM Init
#import "Crosstable.gvl"
#import "Resource1.gvl"

Conf1_node01 :=1;
Conf1_node02 :=1;
Conf1_node03 :=1;
Conf1_node04 :=1;
Conf1_node05 :=1;
Conf1_node06 :=1;
Conf1_node07 :=1;
Conf1_node08 :=1;
Conf1_node09 :=1;
Conf1_node10 :=1;
Conf1_node11 :=1;
Conf1_node12 :=1;
Conf1_node13 :=1;
Conf1_node14 :=1;
Conf1_node15 :=1;
Conf1_node16 :=1;
Conf1_node17 :=1;
Conf1_node18 :=1;
Conf1_node19 :=1;
Conf1_node20 :=1;
Conf1_node21 :=1;
Conf1_node22 :=1;
Conf1_node23 :=1;
Conf1_node24 :=1;

Conf2_node01 :=1;
Conf2_node02 :=1;
Conf2_node03 :=1;
Conf2_node04 :=1;
Conf2_node05 :=1;
Conf2_node06 :=1;
Conf2_node07 :=1;
Conf2_node08 :=1;
Conf2_node09 :=1;
Conf2_node10 :=1;
Conf2_node11 :=1;
Conf2_node12 :=1;
Conf2_node13 :=1;
Conf2_node14 :=1;
Conf2_node15 :=1;
Conf2_node16 :=1;
Conf2_node17 :=1;
Conf2_node18 :=1;
Conf2_node19 :=1;
Conf2_node20 :=1;
Conf2_node21 :=1;
Conf2_node22 :=1;
Conf2_node23 :=1;
Conf2_node24 :=1;

Conf3_node01 :=1;
Conf3_node02 :=1;
Conf3_node03 :=1;
Conf3_node04 :=1;
Conf3_node05 :=1;
Conf3_node06 :=1;
Conf3_node07 :=1;
Conf3_node08 :=1;
Conf3_node09 :=1;
Conf3_node10 :=1;
Conf3_node11 :=1;
Conf3_node12 :=1;
Conf3_node13 :=1;
Conf3_node14 :=1;
Conf3_node15 :=1;
Conf3_node16 :=1;
Conf3_node17 :=1;
Conf3_node18 :=1;
Conf3_node19 :=1;
Conf3_node20 :=1;
Conf3_node21 :=1;
Conf3_node22 :=1;
Conf3_node23 :=1;
Conf3_node24 :=1;

Conf4_node01 :=1;
Conf4_node02 :=1;
Conf4_node03 :=1;
Conf4_node04 :=1;
Conf4_node05 :=1;
Conf4_node06 :=1;
Conf4_node07 :=1;
Conf4_node08 :=1;
Conf4_node09 :=1;
Conf4_node10 :=1;
Conf4_node11 :=1;
Conf4_node12 :=1;
Conf4_node13 :=1;
Conf4_node14 :=1;
Conf4_node15 :=1;
Conf4_node16 :=1;
Conf4_node17 :=1;
Conf4_node18 :=1;
Conf4_node19 :=1;
Conf4_node20 :=1;
Conf4_node21 :=1;
Conf4_node22 :=1;
Conf4_node23 :=1;
Conf4_node24 :=1;

ConfAi1_node01 := 2;
ConfAi1_node02 := 2;
ConfAi1_node03 := 2;
ConfAi1_node04 := 2;
ConfAi1_node05 := 2;
ConfAi1_node06 := 2;
ConfAi1_node07 := 2;
ConfAi1_node08 := 2;
ConfAi1_node09 := 2;
ConfAi1_node10 := 2;
ConfAi1_node11 := 2;
ConfAi1_node12 := 2;
ConfAi1_node13 := 2;
ConfAi1_node14 := 2;
ConfAi1_node15 := 2;
ConfAi1_node16 := 2;
ConfAi1_node17 := 2;
ConfAi1_node18 := 2;
ConfAi1_node19 := 2;
ConfAi1_node20 := 2;
ConfAi1_node21 := 2;
ConfAi1_node22 := 2;
ConfAi1_node23 := 2;
ConfAi1_node24 := 2;

ConfAi2_node01 := 2;
ConfAi2_node02 := 2;
ConfAi2_node03 := 2;
ConfAi2_node04 := 2;
ConfAi2_node05 := 2;
ConfAi2_node06 := 2;
ConfAi2_node07 := 2;
ConfAi2_node08 := 2;
ConfAi2_node09 := 2;
ConfAi2_node10 := 2;
ConfAi2_node11 := 2;
ConfAi2_node12 := 2;
ConfAi2_node13 := 2;
ConfAi2_node14 := 2;
ConfAi2_node15 := 2;
ConfAi2_node16 := 2;
ConfAi2_node17 := 2;
ConfAi2_node18 := 2;
ConfAi2_node19 := 2;
ConfAi2_node20 := 2;
ConfAi2_node21 := 2;
ConfAi2_node22 := 2;
ConfAi2_node23 := 2;
ConfAi2_node24 := 2;

END_PROGRAM

(* ---- Normal.st ---- *)
(*[[
]]*)
PROGRAM Normal
#import "Crosstable.gvl"
#import "Resource1.gvl"
VAR
	counter : uint := 0;
	onoff : bool := true;
	first : bool := true;
	timer : TON;
	value : bool := true;
	timer_ms : UINT := 0;
	do_second_loop : bool := false;

END_VAR

	(* increment timer *)
	timer_ms := timer_ms + 50;

	(* check can status *)
	if CH0_01_NODERUN = false then
		if not first then
			errors_can := errors_can + 1;
		end_if;
 	    return;
	end_if;

	(* init *)
	if first then
		first := false;

		(* 0. init analog outputs *)
		PLC_AnOutConf_1 := 2;
		PLC_AnOutConf_2 := 2;
		PLC_AnOut_1 := 0;
		PLC_AnOut_2 := 0;

		errors_can := 0;

		(* 1. reset latency errors *)
		errors_01 := 0;
		errors_02 := 0;
		errors_03 := 0;
		errors_04 := 0;
		errors_05 := 0;
		errors_06 := 0;
		errors_07 := 0;
		errors_08 := 0;
		errors_09 := 0;
		errors_10 := 0;
		errors_11 := 0;
		errors_12 := 0;
		errors_13 := 0;
		errors_14 := 0;
		errors_15 := 0;
		errors_16 := 0;
		errors_17 := 0;
		errors_18 := 0;
		errors_19 := 0;
		errors_20 := 0;
		errors_21 := 0;
		errors_22 := 0;
		errors_23 := 0;
		errors_24 := 0;

		(* 2. reset latency timer *)
		timer_ms := 0;

		(* 3. reset latencies, ... *)
		latency_01_ms := 0;
		latency_02_ms := 0;
		latency_03_ms := 0;
		latency_04_ms := 0;
		latency_05_ms := 0;
		latency_06_ms := 0;
		latency_07_ms := 0;
		latency_08_ms := 0;
		latency_09_ms := 0;
		latency_10_ms := 0;
		latency_11_ms := 0;
		latency_12_ms := 0;
		latency_13_ms := 0;
		latency_14_ms := 0;
		latency_15_ms := 0;
		latency_16_ms := 0;
		latency_17_ms := 0;
		latency_18_ms := 0;
		latency_19_ms := 0;
		latency_20_ms := 0;
		latency_21_ms := 0;
		latency_22_ms := 0;
		latency_23_ms := 0;
		latency_24_ms := 0;

		min_latency_01_m := 0;
		min_latency_02_m := 0;
		min_latency_03_m := 0;
		min_latency_04_m := 0;
		min_latency_05_m := 0;
		min_latency_06_m := 0;
		min_latency_07_m := 0;
		min_latency_08_m := 0;
		min_latency_09_m := 0;
		min_latency_10_m := 0;
		min_latency_11_m := 0;
		min_latency_12_m := 0;
		min_latency_13_m := 0;
		min_latency_14_m := 0;
		min_latency_15_m := 0;
		min_latency_16_m := 0;
		min_latency_17_m := 0;
		min_latency_18_m := 0;
		min_latency_19_m := 0;
		min_latency_20_m := 0;
		min_latency_21_m := 0;
		min_latency_22_m := 0;
		min_latency_23_m := 0;
		min_latency_24_m := 0;

		max_latency_01_m := 0;
		max_latency_02_m := 0;
		max_latency_03_m := 0;
		max_latency_04_m := 0;
		max_latency_05_m := 0;
		max_latency_06_m := 0;
		max_latency_07_m := 0;
		max_latency_08_m := 0;
		max_latency_09_m := 0;
		max_latency_10_m := 0;
		max_latency_11_m := 0;
		max_latency_12_m := 0;
		max_latency_13_m := 0;
		max_latency_14_m := 0;
		max_latency_15_m := 0;
		max_latency_16_m := 0;
		max_latency_17_m := 0;
		max_latency_18_m := 0;
		max_latency_19_m := 0;
		max_latency_20_m := 0;
		max_latency_21_m := 0;
		max_latency_22_m := 0;
		max_latency_23_m := 0;
		max_latency_24_m := 0;

		(* 4. set first output values *)
		value := true;
		PLC_DigOut_1 := true;
		PLC_AnOut_1 := 900;
		PLC_AnOut_2 := 100;

	end_if;

	timer (IN := true, PT := T#4s);

	(* FIRST/LAST STEP *)
	if timer.q = true then

		(* 0. rearm timer *)
		timer (IN := false);

		(* 1. check latency errors *)
		if latency_01_ms = 0 then
			errors_01 := errors_01 + 1;
		end_if;
		if latency_02_ms = 0 then
			errors_02 := errors_02 + 1;
		end_if;
		if latency_03_ms = 0 then
			errors_03 := errors_03 + 1;
		end_if;
		if latency_04_ms = 0 then
			errors_04 := errors_04 + 1;
		end_if;
		if latency_05_ms = 0 then
			errors_05 := errors_05 + 1;
		end_if;
		if latency_06_ms = 0 then
			errors_06 := errors_06 + 1;
		end_if;
		if latency_07_ms = 0 then
			errors_07 := errors_07 + 1;
		end_if;
		if latency_08_ms = 0 then
			errors_08 := errors_08 + 1;
		end_if;
		if latency_09_ms = 0 then
			errors_09 := errors_09 + 1;
		end_if;
		if latency_10_ms = 0 then
			errors_10 := errors_10 + 1;
		end_if;
		if latency_11_ms = 0 then
			errors_11 := errors_11 + 1;
		end_if;
		if latency_12_ms = 0 then
			errors_12 := errors_12 + 1;
		end_if;
		if latency_13_ms = 0 then
			errors_13 := errors_13 + 1;
		end_if;
		if latency_14_ms = 0 then
			errors_14 := errors_14 + 1;
		end_if;
		if latency_15_ms = 0 then
			errors_15 := errors_15 + 1;
		end_if;
		if latency_16_ms = 0 then
			errors_16 := errors_16 + 1;
		end_if;
		if latency_17_ms = 0 then
			errors_17 := errors_17 + 1;
		end_if;
		if latency_18_ms = 0 then
			errors_18 := errors_18 + 1;
		end_if;
		if latency_19_ms = 0 then
			errors_19 := errors_19 + 1;
		end_if;
		if latency_20_ms = 0 then
			errors_20 := errors_20 + 1;
		end_if;
		if latency_21_ms = 0 then
			errors_21 := errors_21 + 1;
		end_if;
		if latency_22_ms = 0 then
			errors_22 := errors_22 + 1;
		end_if;
		if latency_23_ms = 0 then
			errors_23 := errors_23 + 1;
		end_if;
		if latency_24_ms = 0 then
			errors_24 := errors_24 + 1;
		end_if;

		(* 2. reset latency timer *)
		timer_ms := 0;

		(* 3. reset latencies, ... *)
	    latency_01_ms := 0;
		latency_02_ms := 0;
		latency_03_ms := 0;
		latency_04_ms := 0;
		latency_05_ms := 0;
		latency_06_ms := 0;
		latency_07_ms := 0;
		latency_08_ms := 0;
		latency_09_ms := 0;
		latency_10_ms := 0;
		latency_11_ms := 0;
		latency_12_ms := 0;
		latency_13_ms := 0;
		latency_14_ms := 0;
		latency_15_ms := 0;
		latency_16_ms := 0;
		latency_17_ms := 0;
		latency_18_ms := 0;
		latency_19_ms := 0;
		latency_20_ms := 0;
		latency_21_ms := 0;
		latency_22_ms := 0;
		latency_23_ms := 0;
		latency_24_ms := 0;

		(* 4. set new output value *)
		value := not value;
		PLC_DigOut_1 := value;
		if value then
			PLC_AnOut_1 := 900;
			PLC_AnOut_2 := 100;
		else
			PLC_AnOut_1 := 100;
			PLC_AnOut_2 := 900;
		end_if;

	(* OTHER STEPS *)
	else

		(* for each node: latency from TPAC:DigOut_1 to NODE:DigIn_7 to NODE:DigOut_8 *)

		if latency_01_ms = 0 and DigIn_7_node01 = value then
			(* measure the latency *)
		    latency_01_ms := timer_ms;
			if max_latency_01_m < timer_ms then
				max_latency_01_m := timer_ms;
			end_if;
			if min_latency_01_m > timer_ms or min_latency_01_m = 0 then
				min_latency_01_m := timer_ms;
			end_if;
			(* write the output *)
			DigOut_8_node01 := value;
		end_if;
		if latency_02_ms = 0 and DigIn_7_node02 = value then
			(* measure the latency *)
		    latency_02_ms := timer_ms;
			if max_latency_02_m < timer_ms then
				max_latency_02_m := timer_ms;
			end_if;
			if min_latency_02_m > timer_ms or min_latency_02_m = 0 then
				min_latency_02_m := timer_ms;
			end_if;
			(* write the output *)
			DigOut_8_node02 := value;
		end_if;
		if latency_03_ms = 0 and DigIn_7_node03 = value then
			(* measure the latency *)
		    latency_03_ms := timer_ms;
			if max_latency_03_m < timer_ms then
				max_latency_03_m := timer_ms;
			end_if;
			if min_latency_03_m > timer_ms or min_latency_03_m = 0 then
				min_latency_03_m := timer_ms;
			end_if;
			(* write the output *)
			DigOut_8_node03 := value;
		end_if;
		if latency_04_ms = 0 and DigIn_7_node04 = value then
			(* measure the latency *)
		    latency_04_ms := timer_ms;
			if max_latency_04_m < timer_ms then
				max_latency_04_m := timer_ms;
			end_if;
			if min_latency_04_m > timer_ms or min_latency_04_m = 0 then
				min_latency_04_m := timer_ms;
			end_if;
			(* write the output *)
			DigOut_8_node04 := value;
		end_if;
		if latency_05_ms = 0 and DigIn_7_node05 = value then
			(* measure the latency *)
		    latency_05_ms := timer_ms;
			if max_latency_05_m < timer_ms then
				max_latency_05_m := timer_ms;
			end_if;
			if min_latency_05_m > timer_ms or min_latency_05_m = 0 then
				min_latency_05_m := timer_ms;
			end_if;
			(* write the output *)
			DigOut_8_node05 := value;
		end_if;
		if latency_06_ms = 0 and DigIn_7_node06 = value then
			(* measure the latency *)
		    latency_06_ms := timer_ms;
			if max_latency_06_m < timer_ms then
				max_latency_06_m := timer_ms;
			end_if;
			if min_latency_06_m > timer_ms or min_latency_06_m = 0 then
				min_latency_06_m := timer_ms;
			end_if;
			(* write the output *)
			DigOut_8_node06 := value;
		end_if;
		if latency_07_ms = 0 and DigIn_7_node07 = value then
			(* measure the latency *)
		    latency_07_ms := timer_ms;
			if max_latency_07_m < timer_ms then
				max_latency_07_m := timer_ms;
			end_if;
			if min_latency_07_m > timer_ms or min_latency_07_m = 0 then
				min_latency_07_m := timer_ms;
			end_if;
			(* write the output *)
			DigOut_8_node07 := value;
		end_if;
		if latency_08_ms = 0 and DigIn_7_node08 = value then
			(* measure the latency *)
		    latency_08_ms := timer_ms;
			if max_latency_08_m < timer_ms then
				max_latency_08_m := timer_ms;
			end_if;
			if min_latency_08_m > timer_ms or min_latency_08_m = 0 then
				min_latency_08_m := timer_ms;
			end_if;
			(* write the output *)
			DigOut_8_node08 := value;
		end_if;
		if latency_09_ms = 0 and DigIn_7_node09 = value then
			(* measure the latency *)
		    latency_09_ms := timer_ms;
			if max_latency_09_m < timer_ms then
				max_latency_09_m := timer_ms;
			end_if;
			if min_latency_09_m > timer_ms or min_latency_09_m = 0 then
				min_latency_09_m := timer_ms;
			end_if;
			(* write the output *)
			DigOut_8_node09 := value;
		end_if;
		if latency_10_ms = 0 and DigIn_7_node10 = value then
			(* measure the latency *)
		    latency_10_ms := timer_ms;
			if max_latency_10_m < timer_ms then
				max_latency_10_m := timer_ms;
			end_if;
			if min_latency_10_m > timer_ms or min_latency_10_m = 0 then
				min_latency_10_m := timer_ms;
			end_if;
			(* write the output *)
			DigOut_8_node10 := value;
		end_if;
		if latency_11_ms = 0 and DigIn_7_node11 = value then
			(* measure the latency *)
		    latency_11_ms := timer_ms;
			if max_latency_11_m < timer_ms then
				max_latency_11_m := timer_ms;
			end_if;
			if min_latency_11_m > timer_ms or min_latency_11_m = 0 then
				min_latency_11_m := timer_ms;
			end_if;
			(* write the output *)
			DigOut_8_node11 := value;
		end_if;
		if latency_12_ms = 0 and DigIn_7_node12 = value then
			(* measure the latency *)
		    latency_12_ms := timer_ms;
			if max_latency_12_m < timer_ms then
				max_latency_12_m := timer_ms;
			end_if;
			if min_latency_12_m > timer_ms or min_latency_12_m = 0 then
				min_latency_12_m := timer_ms;
			end_if;
			(* write the output *)
			DigOut_8_node12 := value;
		end_if;
		if latency_13_ms = 0 and DigIn_7_node13 = value then
			(* measure the latency *)
		    latency_13_ms := timer_ms;
			if max_latency_13_m < timer_ms then
				max_latency_13_m := timer_ms;
			end_if;
			if min_latency_13_m > timer_ms or min_latency_13_m = 0 then
				min_latency_13_m := timer_ms;
			end_if;
			(* write the output *)
			DigOut_8_node13 := value;
		end_if;
		if latency_14_ms = 0 and DigIn_7_node14 = value then
			(* measure the latency *)
		    latency_14_ms := timer_ms;
			if max_latency_14_m < timer_ms then
				max_latency_14_m := timer_ms;
			end_if;
			if min_latency_14_m > timer_ms or min_latency_14_m = 0 then
				min_latency_14_m := timer_ms;
			end_if;
			(* write the output *)
			DigOut_8_node14 := value;
		end_if;
		if latency_15_ms = 0 and DigIn_7_node15 = value then
			(* measure the latency *)
		    latency_15_ms := timer_ms;
			if max_latency_15_m < timer_ms then
				max_latency_15_m := timer_ms;
			end_if;
			if min_latency_15_m > timer_ms or min_latency_15_m = 0 then
				min_latency_15_m := timer_ms;
			end_if;
			(* write the output *)
			DigOut_8_node15 := value;
		end_if;
		if latency_16_ms = 0 and DigIn_7_node16 = value then
			(* measure the latency *)
		    latency_16_ms := timer_ms;
			if max_latency_16_m < timer_ms then
				max_latency_16_m := timer_ms;
			end_if;
			if min_latency_16_m > timer_ms or min_latency_16_m = 0 then
				min_latency_16_m := timer_ms;
			end_if;
			(* write the output *)
			DigOut_8_node16 := value;
		end_if;
		if latency_17_ms = 0 and DigIn_7_node17 = value then
			(* measure the latency *)
		    latency_17_ms := timer_ms;
			if max_latency_17_m < timer_ms then
				max_latency_17_m := timer_ms;
			end_if;
			if min_latency_17_m > timer_ms or min_latency_17_m = 0 then
				min_latency_17_m := timer_ms;
			end_if;
			(* write the output *)
			DigOut_8_node17 := value;
		end_if;
		if latency_18_ms = 0 and DigIn_7_node18 = value then
			(* measure the latency *)
		    latency_18_ms := timer_ms;
			if max_latency_18_m < timer_ms then
				max_latency_18_m := timer_ms;
			end_if;
			if min_latency_18_m > timer_ms or min_latency_18_m = 0 then
				min_latency_18_m := timer_ms;
			end_if;
			(* write the output *)
			DigOut_8_node18 := value;
		end_if;
		if latency_19_ms = 0 and DigIn_7_node19 = value then
			(* measure the latency *)
		    latency_19_ms := timer_ms;
			if max_latency_19_m < timer_ms then
				max_latency_19_m := timer_ms;
			end_if;
			if min_latency_19_m > timer_ms or min_latency_19_m = 0 then
				min_latency_19_m := timer_ms;
			end_if;
			(* write the output *)
			DigOut_8_node19 := value;
		end_if;
		if latency_20_ms = 0 and DigIn_7_node20 = value then
			(* measure the latency *)
		    latency_20_ms := timer_ms;
			if max_latency_20_m < timer_ms then
				max_latency_20_m := timer_ms;
			end_if;
			if min_latency_20_m > timer_ms or min_latency_20_m = 0 then
				min_latency_20_m := timer_ms;
			end_if;
			(* write the output *)
			DigOut_8_node20 := value;
		end_if;
		if latency_21_ms = 0 and DigIn_7_node21 = value then
			(* measure the latency *)
		    latency_21_ms := timer_ms;
			if max_latency_21_m < timer_ms then
				max_latency_21_m := timer_ms;
			end_if;
			if min_latency_21_m > timer_ms or min_latency_21_m = 0 then
				min_latency_21_m := timer_ms;
			end_if;
			(* write the output *)
			DigOut_8_node21 := value;
		end_if;
		if latency_22_ms = 0 and DigIn_7_node22 = value then
			(* measure the latency *)
		    latency_22_ms := timer_ms;
			if max_latency_22_m < timer_ms then
				max_latency_22_m := timer_ms;
			end_if;
			if min_latency_22_m > timer_ms or min_latency_22_m = 0 then
				min_latency_22_m := timer_ms;
			end_if;
			(* write the output *)
			DigOut_8_node22 := value;
		end_if;
		if latency_23_ms = 0 and DigIn_7_node23 = value then
			(* measure the latency *)
		    latency_23_ms := timer_ms;
			if max_latency_23_m < timer_ms then
				max_latency_23_m := timer_ms;
			end_if;
			if min_latency_23_m > timer_ms or min_latency_23_m = 0 then
				min_latency_23_m := timer_ms;
			end_if;
			(* write the output *)
			DigOut_8_node23 := value;
		end_if;
		if latency_24_ms = 0 and DigIn_7_node24 = value then
			(* measure the latency *)
		    latency_24_ms := timer_ms;
			if max_latency_24_m < timer_ms then
				max_latency_24_m := timer_ms;
			end_if;
			if min_latency_24_m > timer_ms or min_latency_24_m = 0 then
				min_latency_24_m := timer_ms;
			end_if;
			(* write the output *)
			DigOut_8_node24 := value;
		end_if;

	end_if;

	if do_second_loop then
		(* one round true and one round false *)
		onoff := ((counter / 12) mod 2) = 0;

		(* in each round touch every node *)
		case (counter mod 12) + 1 of
			1: DigOut_5_node01 := onoff; DigOut_5_node13 := onoff;
		    2: DigOut_5_node02 := onoff; DigOut_5_node14 := onoff;
	        3: DigOut_5_node03 := onoff; DigOut_5_node15 := onoff;
		    4: DigOut_5_node04 := onoff; DigOut_5_node16 := onoff;
		    5: DigOut_5_node05 := onoff; DigOut_5_node17 := onoff;
		    6: DigOut_5_node06 := onoff; DigOut_5_node18 := onoff;
		    7: DigOut_5_node07 := onoff; DigOut_5_node19 := onoff;
		    8: DigOut_5_node08 := onoff; DigOut_5_node20 := onoff;
		    9: DigOut_5_node09 := onoff; DigOut_5_node21 := onoff;
		   10: DigOut_5_node10 := onoff; DigOut_5_node22 := onoff;
		   11: DigOut_5_node11 := onoff; DigOut_5_node23 := onoff;
		   12: DigOut_5_node12 := onoff; DigOut_5_node24 := onoff;
	    else
		   ;
		end_case;

		(* increment the counter, with overflow *)
		counter := counter + 1;

	end_if;

END_PROGRAM

(* ---- Slow.st ---- *)
(*[[
]]*)
PROGRAM Slow
#import "Crosstable.gvl"
#import "Resource1.gvl"

	PLC_DigOut_1 := not PLC_DigOut_1;

END_PROGRAM
